// TIA Portal project "HW_2100068_montaz_menica_PSA_8HP_EL58_V18" (V18)

(* hardware
DEVICE "GSD device_8"  GSD.Device.PN
   slot 0: "vitc06a"  EX600-SPN#  EX600-SPN#
      slot 0: "EX600-SPN#"  EX600-SPN#
      slot 1: "Interface"  Interface
         slot 1: "Port 1"  Port 1
         slot 2: "Port 2"  Port 2
   slot 0: "Rack"  Rack  V1.0
   slot 1: "EX600-DX#D_1"  EX600-DX#D  EX600-DX#D
      slot 0: "EX600-DX#D"  EX600-DX#D
   slot 2: "EX600-DY#B_1"  EX600-DY#B  EX600-DY#B
      slot 0: "EX600-DY#B"  EX600-DY#B
   slot 3: "EX600-AXA_1"  EX600-AXA  EX600-AXA
      slot 0: "EX600-AXA"  EX600-AXA
   slot 4: "EX600-SPN (32 coils)_1"  EX600-SPN (32 coils)  EX600-SPN
      slot 0: "EX600-SPN"  EX600-SPN
DEVICE "GSD device_7"  GSD.Device.PN
   slot 0: "vitc04e"  EX600-SPN#  EX600-SPN#
      slot 0: "EX600-SPN#"  EX600-SPN#
      slot 1: "Interface"  Interface
         slot 1: "Port 1"  Port 1
         slot 2: "Port 2"  Port 2
   slot 0: "Rack"  Rack  V1.0
   slot 1: "EX600-DX#D_1"  EX600-DX#D  EX600-DX#D
      slot 0: "EX600-DX#D"  EX600-DX#D
   slot 2: "EX600-DY#B_1"  EX600-DY#B  EX600-DY#B
      slot 0: "EX600-DY#B"  EX600-DY#B
   slot 3: "EX600-AXA_1"  EX600-AXA  EX600-AXA
      slot 0: "EX600-AXA"  EX600-AXA
   slot 4: "EX600-SPN (32 coils)_1"  EX600-SPN (32 coils)  EX600-SPN
      slot 0: "EX600-SPN"  EX600-SPN
DEVICE "GSD device_3"  GSD.Device.PN
   slot 0: "mtstc10c"  SR-LR1  SR-LR1  1.0
      slot 0: "SR-LR1"  SR-LR1  1.0
      slot 1: "Interface"  Interface
         slot 1: "Port 1"  Port 1
   slot 0: "Rack"  Rack  V1.0
   slot 1: "Handshake and General Error Status Bits_1"  Handshake and General Error Status Bits
      slot 0: "Handshake and General Error Status Bits"  Handshake and General Error Status Bits
   slot 3: "Completion Status Bits_1"  Completion Status Bits
      slot 0: "Completion Status Bits"  Completion Status Bits
   slot 5: "Terminal Status Bits_1"  Terminal Status Bits
      slot 0: "Terminal Status Bits"  Terminal Status Bits
   slot 8: "Operation Result Status_1"  Operation Result Status
      slot 0: "Operation Result Status"  Operation Result Status
   slot 9: "Read Data 128Byte_1"  Read Data 128Byte
      slot 0: "Read Data 128Byte"  Read Data 128Byte
   slot 10: "Latch and Error Clear Control Bits_1"  Latch and Error Clear Control Bits
      slot 0: "Latch and Error Clear Control Bits"  Latch and Error Clear Control Bits
   slot 12: "Completion Clear Control Bits_1"  Completion Clear Control Bits
      slot 0: "Completion Clear Control Bits"  Completion Clear Control Bits
DEVICE "GSD device_11"  GSD.Device.PN
   slot 0: "mtstc10a"  KRC4-ProfiNet_3.2  V3.2
      slot 0: "KRC4-ProfiNet_3.2"  KRC4-ProfiNet_3.2
      slot 1: "Interface1"  Interface1
         slot 1: "Port1"  Port1
   slot 0: "Rack"  Rack  V1.0
   slot 1: "64 safe digital in- and outputs_1"  64 safe digital in- and outputs  KUKA KR C4 Device FIO64
      slot 0: "64 safe digital in- and outputs"  64 safe digital in- and outputs
   slot 2: "256 digital in- and outputs_1"  256 digital in- and outputs  KUKA KR C4 Device IO256
      slot 0: "256 digital in- and outputs"  256 digital in- and outputs
DEVICE "GSD device_18"  GSD.Device
   slot 0: "mtstc07b"  6ES7 158-0AD01-0XA0  B0
   slot 0: "Rack_0"  Rail
DEVICE "GSD device_20"  GSD.Device.PN
   slot 0: "mtstc07a"  NIC 52-RE/PNS V2.0 - V2.x  1544.100  V2.x
      slot 0: "NIC 52-RE/PNS V2.0 - V2.x"  NIC 52-RE/PNS V2.0 - V2.x
      slot 1: "PN-IO"  PN-IO
         slot 1: "Port 1"  Port 1
         slot 2: "Port 2"  Port 2
   slot 0: "Rack"  Rack  V1.0
   slot 1: "1 Unsigned32 Output_1"  1 Unsigned32 Output
      slot 0: "1 Unsigned32 Output"  1 Unsigned32 Output
   slot 2: "64 Bytes Output_1"  64 Bytes Output
      slot 0: "64 Bytes Output"  64 Bytes Output
   slot 5: "1 Unsigned32 Input_1"  1 Unsigned32 Input
      slot 0: "1 Unsigned32 Input"  1 Unsigned32 Input
   slot 6: "64 Bytes Input_1"  64 Bytes Input
      slot 0: "64 Bytes Input"  64 Bytes Input
DEVICE "GSD device_2"  GSD.Device.PN
   slot 0: "mtstc06c"  SR-LR1  SR-LR1  1.0
      slot 0: "SR-LR1"  SR-LR1  1.0
      slot 1: "Interface"  Interface
         slot 1: "Port 1"  Port 1
   slot 0: "Rack"  Rack  V1.0
   slot 1: "Handshake and General Error Status Bits_1"  Handshake and General Error Status Bits
      slot 0: "Handshake and General Error Status Bits"  Handshake and General Error Status Bits
   slot 3: "Completion Status Bits_1"  Completion Status Bits
      slot 0: "Completion Status Bits"  Completion Status Bits
   slot 5: "Terminal Status Bits_1"  Terminal Status Bits
      slot 0: "Terminal Status Bits"  Terminal Status Bits
   slot 8: "Operation Result Status_1"  Operation Result Status
      slot 0: "Operation Result Status"  Operation Result Status
   slot 9: "Read Data 128Byte_1"  Read Data 128Byte
      slot 0: "Read Data 128Byte"  Read Data 128Byte
   slot 10: "Latch and Error Clear Control Bits_1"  Latch and Error Clear Control Bits
      slot 0: "Latch and Error Clear Control Bits"  Latch and Error Clear Control Bits
   slot 12: "Completion Clear Control Bits_1"  Completion Clear Control Bits
      slot 0: "Completion Clear Control Bits"  Completion Clear Control Bits
DEVICE "GSD device_10"  GSD.Device.PN
   slot 0: "mtstc06a"  KRC4-ProfiNet_3.2  V3.2
      slot 0: "KRC4-ProfiNet_3.2"  KRC4-ProfiNet_3.2
      slot 1: "Interface1"  Interface1
         slot 1: "Port1"  Port1
   slot 0: "Rack"  Rack  V1.0
   slot 1: "64 safe digital in- and outputs_1"  64 safe digital in- and outputs  KUKA KR C4 Device FIO64
      slot 0: "64 safe digital in- and outputs"  64 safe digital in- and outputs
   slot 2: "256 digital in- and outputs_1"  256 digital in- and outputs  KUKA KR C4 Device IO256
      slot 0: "256 digital in- and outputs"  256 digital in- and outputs
DEVICE "GSD device_17"  GSD.Device
   slot 0: "mtstc05"  6ES7 158-0AD01-0XA0  B0
   slot 0: "Rack_0"  Rail
DEVICE "GSD device_16"  GSD.Device.PN
   slot 0: "mtstc04e"  KRC4-ProfiNet_3.2  V3.2
      slot 0: "KRC4-ProfiNet_3.2"  KRC4-ProfiNet_3.2
      slot 1: "Interface1"  Interface1
         slot 1: "Port1"  Port1
   slot 0: "Rack"  Rack  V1.0
   slot 1: "64 safe digital in- and outputs_1"  64 safe digital in- and outputs  KUKA KR C4 Device FIO64
      slot 0: "64 safe digital in- and outputs"  64 safe digital in- and outputs
   slot 2: "256 digital in- and outputs_1"  256 digital in- and outputs  KUKA KR C4 Device IO256
      slot 0: "256 digital in- and outputs"  256 digital in- and outputs
DEVICE "GSD device_15"  GSD.Device
   slot 0: "mtstc04b"  6ES7 158-0AD01-0XA0  B0
   slot 0: "Rack_0"  Rail
DEVICE "ET 200SP station_2"  ET 200SP-Station
   slot 0: "et200sptc10a"  IM 155-6 PN ST  6ES7 155-6AU00-0BN0  V3.3
   slot 0: "Rack_0"  Rack  6ES5 710-8MAx1
   slot 1: "111A2 DI 16x24_1"  DI 16x24VDC ST  6ES7 131-6BH00-0BA0  V1.1
      slot 1: "111A2 DI 16x24_1"  DI 16x24VDC ST
   slot 2: "111A3 DI 16x24_2"  DI 16x24VDC ST  6ES7 131-6BH00-0BA0  V1.1
      slot 1: "111A3 DI 16x24_2"  DI 16x24VDC ST
   slot 3: "112A1 DQ 16x24_1"  DQ 16x24VDC/0.5A ST  6ES7 132-6BH00-0BA0  V1.1
      slot 1: "112A1 DQ 16x24_1"  DQ 16x24VDC/0.5A ST
   slot 4: "112A2 DQ 16x24_2"  DQ 16x24VDC/0.5A ST  6ES7 132-6BH00-0BA0  V1.1
      slot 1: "112A2 DQ 16x24_2"  DQ 16x24VDC/0.5A ST
   slot 5: "112A3 DQ 16x24_3"  DQ 16x24VDC/0.5A ST  6ES7 132-6BH00-0BA0  V1.1
      slot 1: "112A3 DQ 16x24_3"  DQ 16x24VDC/0.5A ST
   slot 6: "Server module_1"  Server module  6ES7 193-6PA00-0AA0  V1.1
      slot 1: "Server module_1"  Server module
   slot 127: "BA 2xRJ45"  BA 2xRJ45  6ES7 193-6AR00-0AA0  V0.0
      slot 1: "Port_1"  X1 P1 R  6ES7 193-6AR00-0AA0  V0.0
      slot 2: "Port_2"  X1 P2 R  6ES7 193-6AR00-0AA0  V0.0
DEVICE "ET 200SP station_4"  ET 200SP-Station
   slot 0: "et200sptc06a"  IM 155-6 PN ST  6ES7 155-6AU00-0BN0  V3.3
   slot 0: "Rack_0"  Rack  6ES5 710-8MAx1
   slot 1: "111A2 DI 16x24_1"  DI 16x24VDC ST  6ES7 131-6BH00-0BA0  V1.1
      slot 1: "111A2 DI 16x24_1"  DI 16x24VDC ST
   slot 2: "111A3 DI 16x24_2"  DI 16x24VDC ST  6ES7 131-6BH00-0BA0  V1.1
      slot 1: "111A3 DI 16x24_2"  DI 16x24VDC ST
   slot 3: "112A1 DQ 16x24_1"  DQ 16x24VDC/0.5A ST  6ES7 132-6BH00-0BA0  V1.1
      slot 1: "112A1 DQ 16x24_1"  DQ 16x24VDC/0.5A ST
   slot 4: "112A2 DQ 16x24_2"  DQ 16x24VDC/0.5A ST  6ES7 132-6BH00-0BA0  V1.1
      slot 1: "112A2 DQ 16x24_2"  DQ 16x24VDC/0.5A ST
   slot 5: "112A3 DQ 16x24_3"  DQ 16x24VDC/0.5A ST  6ES7 132-6BH00-0BA0  V1.1
      slot 1: "112A3 DQ 16x24_3"  DQ 16x24VDC/0.5A ST
   slot 6: "Server module_1"  Server module  6ES7 193-6PA00-0AA0  V1.1
      slot 1: "Server module_1"  Server module
   slot 127: "BA 2xRJ45"  BA 2xRJ45  6ES7 193-6AR00-0AA0  V0.0
      slot 1: "Port_1"  X1 P1 R  6ES7 193-6AR00-0AA0  V0.0
      slot 2: "Port_2"  X1 P2 R  6ES7 193-6AR00-0AA0  V0.0
DEVICE "ET 200SP station_1"  ET 200SP-Station
   slot 0: "et200sp_111a1"  IM 155-6 PN ST  6ES7 155-6AU00-0BN0  V3.3
   slot 0: "Rack_0"  Rack  6ES5 710-8MAx1
   slot 1: "111A2 DI 16x24_1"  DI 16x24VDC ST  6ES7 131-6BH00-0BA0  V1.1
      slot 1: "111A2 DI 16x24_1"  DI 16x24VDC ST
   slot 2: "111A3 DI 16x24_2"  DI 16x24VDC ST  6ES7 131-6BH00-0BA0  V1.1
      slot 1: "111A3 DI 16x24_2"  DI 16x24VDC ST
   slot 3: "111A4 DI 16x24_3"  DI 16x24VDC ST  6ES7 131-6BH00-0BA0  V1.1
      slot 1: "111A4 DI 16x24_3"  DI 16x24VDC ST
   slot 4: "112A1 DQ 16x24_1"  DQ 16x24VDC/0.5A ST  6ES7 132-6BH00-0BA0  V1.1
      slot 1: "112A1 DQ 16x24_1"  DQ 16x24VDC/0.5A ST
   slot 5: "112A2 DQ 16x24_2"  DQ 16x24VDC/0.5A ST  6ES7 132-6BH00-0BA0  V1.1
      slot 1: "112A2 DQ 16x24_2"  DQ 16x24VDC/0.5A ST
   slot 6: "112A3 DQ 16x24_3"  DQ 16x24VDC/0.5A ST  6ES7 132-6BH00-0BA0  V1.1
      slot 1: "112A3 DQ 16x24_3"  DQ 16x24VDC/0.5A ST
   slot 7: "Server module_1"  Server module  6ES7 193-6PA00-0AA0  V1.1
      slot 1: "Server module_1"  Server module
   slot 127: "BA 2xRJ45"  BA 2xRJ45  6ES7 193-6AR00-0AA0  V0.0
      slot 1: "Port_1"  X1 P1 R  6ES7 193-6AR00-0AA0  V0.0
      slot 2: "Port_2"  X1 P2 R  6ES7 193-6AR00-0AA0  V0.0
DEVICE "GSD device_9"  GSD.Device.PN
   slot 0: "Rack"  Rack  V1.0
   slot 0: "vitc10a"  EX600-SPN#  EX600-SPN#
      slot 0: "EX600-SPN#"  EX600-SPN#
      slot 1: "Interface"  Interface
         slot 1: "Port 1"  Port 1
         slot 2: "Port 2"  Port 2
   slot 1: "EX600-DX#D_1"  EX600-DX#D  EX600-DX#D
      slot 0: "EX600-DX#D"  EX600-DX#D
   slot 2: "EX600-DY#B_1"  EX600-DY#B  EX600-DY#B
      slot 0: "EX600-DY#B"  EX600-DY#B
   slot 3: "EX600-AXA_1"  EX600-AXA  EX600-AXA
      slot 0: "EX600-AXA"  EX600-AXA
   slot 4: "EX600-SPN (32 coils)_1"  EX600-SPN (32 coils)  EX600-SPN
      slot 0: "EX600-SPN"  EX600-SPN
DEVICE "GSD device_19"  GSD.Device.PN
   slot 0: "Rack"  Rack  V1.0
   slot 0: "mtstc07b_data"  NIC 52-RE/PNS V2.0 - V2.x  1544.100  V2.x
      slot 0: "NIC 52-RE/PNS V2.0 - V2.x"  NIC 52-RE/PNS V2.0 - V2.x
      slot 1: "PN-IO"  PN-IO
         slot 1: "Port 1"  Port 1
         slot 2: "Port 2"  Port 2
   slot 1: "1 Unsigned32 Output_1"  1 Unsigned32 Output
      slot 0: "1 Unsigned32 Output"  1 Unsigned32 Output
   slot 2: "64 Bytes Output_1"  64 Bytes Output
      slot 0: "64 Bytes Output"  64 Bytes Output
   slot 5: "1 Unsigned32 Input_1"  1 Unsigned32 Input
      slot 0: "1 Unsigned32 Input"  1 Unsigned32 Input
   slot 6: "64 Bytes Input_1"  64 Bytes Input
      slot 0: "64 Bytes Input"  64 Bytes Input
DEVICE "GSD device_12"  GSD.Device.PN
   slot 0: "Rack"  Rack  V1.0
   slot 0: "mtstc07c"  NIC 52-RE/PNS V2.0 - V2.x  1544.100  V2.x
      slot 0: "NIC 52-RE/PNS V2.0 - V2.x"  NIC 52-RE/PNS V2.0 - V2.x
      slot 1: "PN-IO"  PN-IO
         slot 1: "Port 1"  Port 1
         slot 2: "Port 2"  Port 2
   slot 1: "1 Unsigned32 Output_1"  1 Unsigned32 Output
      slot 0: "1 Unsigned32 Output"  1 Unsigned32 Output
   slot 2: "64 Bytes Output_1"  64 Bytes Output
      slot 0: "64 Bytes Output"  64 Bytes Output
   slot 5: "1 Unsigned32 Input_1"  1 Unsigned32 Input
      slot 0: "1 Unsigned32 Input"  1 Unsigned32 Input
   slot 6: "64 Bytes Input_1"  64 Bytes Input
      slot 0: "64 Bytes Input"  64 Bytes Input
DEVICE "GSD device_1"  GSD.Device.PN
   slot 0: "Rack"  Rack  V1.0
   slot 1: "plc_tc04d"  PLC_tc04d  6ES7 512-1SK01-0AB0  V2.8
      slot 0: "Line_To_Cu1"  Line_To_Cu1
      slot 1: "Cu1_To_Line"  Cu1_To_Line
      slot 2: "F_Line_To_Cu1"  F_Line_To_Cu1
      slot 3: "01_SYSTEM_GENERATED_F-CD"  01_SYSTEM_GENERATED_F-CD
      slot 4: "F_CU1_To_Line"  F_CU1_To_Line
      slot 5: "02_SYSTEM_GENERATED_F-CD"  02_SYSTEM_GENERATED_F-CD
      slot 6: "Interface"  Interface
         slot 1: "Port 1"  Port 1
         slot 2: "Port 2"  Port 2
         slot 3: "Port 3"  Port 3
DEVICE "GSD device_4"  GSD.Device.PN
   slot 0: "Rack"  Rack  V1.0
   slot 1: "plc_tc08"  PLC_tc08  6ES7 512-1SK01-0AB0  V2.8
      slot 0: "Line_To_Cu1"  Line_To_Cu1
      slot 1: "Cu1_To_Line"  Cu1_To_Line
      slot 2: "F_Line_To_Cu1"  F_Line_To_Cu1
      slot 3: "01_SYSTEM_GENERATED_F-CD"  01_SYSTEM_GENERATED_F-CD
      slot 4: "F_CU1_To_Line"  F_CU1_To_Line
      slot 5: "02_SYSTEM_GENERATED_F-CD"  02_SYSTEM_GENERATED_F-CD
      slot 6: "Interface"  Interface
         slot 1: "Port 1"  Port 1
         slot 2: "Port 2"  Port 2
         slot 3: "Port 3"  Port 3
DEVICE "GSD device_21"  GSD.Device.PN
   slot 0: "Rack"  Rack  V1.0
   slot 1: "plc_tc11_cd"  PLC_tc11_cd  6ES7 512-1SK01-0AB0  V2.8
      slot 0: "Line_To_Cu1"  Line_To_Cu1
      slot 1: "Cu1_To_Line"  Cu1_To_Line
      slot 2: "F_Line_To_Cu1"  F_Line_To_Cu1
      slot 3: "01_SYSTEM_GENERATED_F-CD"  01_SYSTEM_GENERATED_F-CD
      slot 4: "F_CU1_To_Line"  F_CU1_To_Line
      slot 5: "02_SYSTEM_GENERATED_F-CD"  02_SYSTEM_GENERATED_F-CD
      slot 6: "Line_To_Cu2"  Line_To_Cu2
      slot 7: "Cu2_To_Line"  Cu2_To_Line
      slot 8: "F_Line_To_Cu2"  F_Line_To_Cu2
      slot 9: "03_SYSTEM_GENERATED_F-CD"  03_SYSTEM_GENERATED_F-CD
      slot 10: "F_CU2_To_Line"  F_CU2_To_Line
      slot 11: "04_SYSTEM_GENERATED_F-CD"  04_SYSTEM_GENERATED_F-CD
      slot 12: "Cu3_To_Line"  Cu3_To_Line
      slot 13: "Line_To_Cu3"  Line_To_Cu3
      slot 14: "Interface"  Interface
         slot 1: "Port 1"  Port 1
         slot 2: "Port 2"  Port 2
         slot 3: "Port 3"  Port 3
DEVICE "GSD device_13"  GSD.Device.PN
   slot 0: "Rack"  Rack  V1.0
   slot 1: "plcr1_110a2"  plcr1.112_X1  6ES7 516-3FN02-0AB0  V2.8
      slot 0: "Robot1_ToLine"  Robot1_ToLine
      slot 1: "LineToRobot1"  LineToRobot1
      slot 2: "Robot2_ToLine"  Robot2_ToLine
      slot 3: "LineToRobot2"  LineToRobot2
      slot 4: "Robot3_ToLine"  Robot3_ToLine
      slot 5: "LineToRobot3"  LineToRobot3
      slot 6: "Robot4_ToLine"  Robot4_ToLine
      slot 7: "LineToRobot4"  LineToRobot4
      slot 8: "LineToFLineSafety"  LineToFLineSafety
      slot 9: "FLineToLineSafety"  FLineToLineSafety
      slot 10: "TC09_ToLine"  TC09_ToLine
      slot 11: "LineToTC09"  LineToTC09
      slot 12: "Interface"  Interface
         slot 1: "Port 1"  Port 1
         slot 2: "Port 2"  Port 2
DEVICE "GSD device_14"  GSD.Device.PN
   slot 0: "Rack"  Rack  V1.0
   slot 0: "pnpn_tc11a"  PN/PN Coupler X2  6ES7 158-3AD01-0XA0  V03.00.00
      slot 0: "PN/PN Coupler X2"  PN/PN Coupler X2
      slot 1: "PN-IO-02"  PN-IO-02
         slot 1: "Port 1"  Port 1
         slot 2: "Port 2"  Port 2
   slot 1: "FDI/FDO_6Bytes/12Bytes"  IN/OUT 6 Bytes / 12 Bytes
      slot 0: "IN/OUT 6 Bytes / 12 Bytes"  IN/OUT 6 Bytes / 12 Bytes
   slot 2: "FDI/FDO_12Bytes/6Bytes"  IN/OUT 12 Bytes / 6 Bytes
      slot 0: "IN/OUT 12 Bytes / 6 Bytes"  IN/OUT 12 Bytes / 6 Bytes
   slot 3: "IN  64 Bytes"  IN  64 Bytes
      slot 0: "IN  64 Bytes"  IN  64 Bytes
   slot 4: "OUT  64 Bytes"  OUT  64 Bytes
      slot 0: "OUT  64 Bytes"  OUT  64 Bytes
   slot 5: "IN  64 Bytes_1"  IN  64 Bytes
      slot 0: "IN  64 Bytes"  IN  64 Bytes
DEVICE "pnpn_tc11b"  PnPn.Device
   slot 0: "Rack"  Rail  1.0
   slot 0: "pnpn_tc11b.X1"  PN/PN Coupler  6ES7 158-3AD10-0XA0  V4.2
   slot 1: "pnpn_tc11b.X2"  PN/PN Coupler  6ES7 158-3AD10-0XA0  V4.2
   slot 127: "BA 2xRJ45"  BA 2xRJ45  6ES7 193-6AR00-0AA0  V0.0
      slot 1: "Port_1"  X1 P1 R  6ES7 193-6AR00-0AA0  V0.0
      slot 2: "Port_2"  X1 P2 R  6ES7 193-6AR00-0AA0  V0.0
   slot 127: "BA 2xRJ45"  BA 2xRJ45  6ES7 193-6AR00-0AA0  V0.0
      slot 1: "Port_1"  X2 P1 R  6ES7 193-6AR00-0AA0  V0.0
      slot 2: "Port_2"  X2 P2 R  6ES7 193-6AR00-0AA0  V0.0
DEVICE "GSD device_43"  GSD.Device.PN
   slot 0: "Rack"  Rack  V1.0
   slot 0: "vitc11f"  EX600-SPN#  EX600-SPN#
      slot 0: "EX600-SPN#"  EX600-SPN#
      slot 1: "Interface"  Interface
         slot 1: "Port 1"  Port 1
         slot 2: "Port 2"  Port 2
   slot 1: "EX600-DX#D_1"  EX600-DX#D  EX600-DX#D
      slot 0: "EX600-DX#D"  EX600-DX#D
   slot 2: "EX600-DY#B_1"  EX600-DY#B  EX600-DY#B
      slot 0: "EX600-DY#B"  EX600-DY#B
   slot 3: "EX600-AXA_1"  EX600-AXA  EX600-AXA
      slot 0: "EX600-AXA"  EX600-AXA
   slot 4: "EX600-SPN (32 coils)_1"  EX600-SPN (32 coils)  EX600-SPN
      slot 0: "EX600-SPN"  EX600-SPN
DEVICE "GSD device_42"  GSD.Device.PN
   slot 0: "Rack"  Rack  V1.0
   slot 0: "mtstc11f"  KRC4-ProfiNet_3.2  V3.2
      slot 0: "KRC4-ProfiNet_3.2"  KRC4-ProfiNet_3.2
      slot 1: "Interface1"  Interface1
         slot 1: "Port1"  Port1
   slot 1: "64 safe digital in- and outputs_1"  64 safe digital in- and outputs  KUKA KR C4 Device FIO64
      slot 0: "64 safe digital in- and outputs"  64 safe digital in- and outputs
   slot 2: "256 digital in- and outputs_1"  256 digital in- and outputs  KUKA KR C4 Device IO256
      slot 0: "256 digital in- and outputs"  256 digital in- and outputs
DEVICE "SCALANCE W access point"  SCALANCE W-Station
   slot 0: "SCALANCE W rack"  Rail
   slot 0: "309k1_ap"  SCALANCE W 774-1 RJ45  6GK5 774-1FX00-0AA0  V6.1
DEVICE "SCALANCE XC-200"  SCALANCE X-Station
   slot 0: "SCALANCE X rack"  Rail
   slot 0: "swr1_104s1"  SCALANCE XC224  6GK5 224-0BA00-2AC2  V2.1
DEVICE "S71500/ET200MP station_1"  S7-1500 station
   slot 0: "Rail_0"  Rack  6ES7 590-1***0-0AA0
   slot 1: "plcr1_110a1"  CPU 1516F-3 PN/DP  6ES7 516-3FN01-0AB0  V2.1
      slot 3: "CPU display_1"  6ES7591-1BA00-0AA0
      slot 32768: "PROFINET interface_1"  X1
         slot 32769: "Port_1"  X1 P1
         slot 32770: "Port_2"  X1 P2
      slot 33024: "PROFINET interface_2"  X2
         slot 33025: "Port_1"  X2 P1
      slot 33280: "DP interface_1"  X3
DEVICE "GSD device_5"  GSD.Device.PN
   slot 0: "Rack"  Rack  V1.0
   slot 1: "310a1_plc.profinet interface_1"  310A1_PLC_X1  6ES7 516-3FN01-0AB0  V2.1
      slot 0: "Outputs"  Outputs
      slot 1: "Inputs"  Inputs
      slot 2: "DataToMainLine"  DataToMainLine
      slot 3: "Interface"  Interface
         slot 1: "Port 1"  Port 1
         slot 2: "Port 2"  Port 2
*)

// ===== PLC "plcr1_110a1"  CPU 1516F-3 PN/DP =====

VAR_GLOBAL   // PLC tag table "Default tag table"
   "Clock_Byte" AT %MB0 : Byte;
   "Clock_10Hz" AT %M0.0 : Bool;
   "Clock_5Hz" AT %M0.1 : Bool;
   "Clock_2.5Hz" AT %M0.2 : Bool;
   "Clock_2Hz" AT %M0.3 : Bool;
   "Clock_1.25Hz" AT %M0.4 : Bool;
   "Clock_1Hz" AT %M0.5 : Bool;
   "Clock_0.625Hz" AT %M0.6 : Bool;
   "Clock_0.5Hz" AT %M0.7 : Bool;
   "System_Byte" AT %MB1 : Byte;
   "FirstScan" AT %M1.0 : Bool;
   "DiagStatusUpdate" AT %M1.1 : Bool;
   "AlwaysTRUE" AT %M1.2 : Bool;
   "AlwaysFALSE" AT %M1.3 : Bool;
   "i_161B8_neg" AT %I381.2 : Bool;   // TC04C1_PartPresence
   "i2026.4" AT %I2026.4 : Bool;
   "iW604" AT %IW604 : Int;
   "i171B5" AT %I480.4 : Bool;
   "q_Conveyor" AT %Q1101.7 : Bool;
   "i111A3_9" AT %I483.1 : Bool;
   "i111A3_12" AT %I483.4 : Bool;
   "i2027.4" AT %I2027.4 : Bool;
   "q484.1" AT %Q484.1 : Bool;
   "q484.0" AT %Q484.0 : Bool;
   "iFrictionMoment" AT %IW2058 : Word;
   "i111A3_6" AT %I482.6 : Bool;
   "i111A3_13" AT %I483.5 : Bool;
   "q601.0" AT %Q601.0 : Bool;
   "i600.2" AT %I600.2 : Bool;
   "q384.1" AT %Q384.1 : Bool;
   "i601.1" AT %I601.1 : Bool;
   "i111A3_5" AT %I482.5 : Bool;
   "Q2900_7" AT %Q2900.7 : Bool;
   "i2026.0" AT %I2026.0 : Bool;
   "Tag_1" AT %Q134.1 : Bool;
   "ib2024" AT %IB2024 : Byte;
   "q480.0" AT %Q480.0 : Bool;
   "i2027.1" AT %I2027.1 : Bool;
   "i111A3_4" AT %I482.4 : Bool;
   "i2026.2" AT %I2026.2 : Bool;
   "i111A3_7" AT %I482.7 : Bool;
   "q384.0" AT %Q384.0 : Bool;
   "i171B1" AT %I480.0 : Bool;
   "i171B3" AT %I480.2 : Bool;
   "i111A3_3" AT %I482.3 : Bool;
   "i_161B7" AT %I380.6 : Bool;
   "q600.0" AT %Q600.0 : Bool;
   "q601.2" AT %Q601.2 : Bool;
   "Q2900_6" AT %Q2900.6 : Bool;
   "i600.0" AT %I600.0 : Bool;
   "qTC04B_OutputByte0" AT %QB500 : Byte;
   "i111A3_10" AT %I483.2 : Bool;
   "i172SB2" AT %I481.1 : Bool;
   "i601.0" AT %I601.0 : Bool;
   "Q2900_4" AT %Q2900.4 : Bool;
   "i111A3_8" AT %I483.0 : Bool;
   "ib2025" AT %IB2025 : Byte;
   "Tag_5" AT %Q1105.7 : Bool;
   "i111A3_2" AT %I482.2 : Bool;
   "Q2900_5" AT %Q2900.5 : Bool;
   "i601.3" AT %I601.3 : Bool;
   "i2027.2" AT %I2027.2 : Bool;
   "i111A3_14" AT %I483.6 : Bool;
   "i2027.0" AT %I2027.0 : Bool;
   "i111A3_0" AT %I482.0 : Bool;
   "q600.1" AT %Q600.1 : Bool;
   "i600.3" AT %I600.3 : Bool;
   "i2026.3" AT %I2026.3 : Bool;
   "i171B2" AT %I480.1 : Bool;
   "q600.2" AT %Q600.2 : Bool;
   "qRobotOutOfArea" AT %Q50.7 : Bool;
   "qTC04B_OutputByte1" AT %QB501 : Byte;
   "i171B4" AT %I480.3 : Bool;
   "i171B6" AT %I480.5 : Bool;
   "i2027.3" AT %I2027.3 : Bool;
   "i_161B7_neg" AT %I381.3 : Bool;   // TC04C2_PartPresence
   "Tag_4" AT %I451.0 : Bool;
   "iw602" AT %IW602 : Int;
   "i172SB1" AT %I481.0 : Bool;
   "i_161B8" AT %I380.7 : Bool;
   "i600.1" AT %I600.1 : Bool;
   "i2026.1" AT %I2026.1 : Bool;
   "i601.2" AT %I601.2 : Bool;
   "q482.0" AT %Q482.0 : Bool;
   "q482.1" AT %Q482.1 : Bool;
   "i111A3_15" AT %I483.7 : Bool;
   "fdi_plcr1_110a2_1byte_pnpn" AT %IB116 : Byte;   // z pnpn plcr1_110a2 :
   "iW606" AT %IW606 : Int;
   "i111A3_1" AT %I482.1 : Bool;
   "fdiEstopTC08_Profisafe" AT %I1892.0 : Bool;   // Estop TC08 -Plnenie olejom EMP
   "i111A3_11" AT %I483.3 : Bool;
   "qGreenConveyor(1)" AT %Q480.5 : Bool;
   "qRedRework(1)" AT %Q480.2 : Bool;
   "qGreenRework(1)" AT %Q480.3 : Bool;
   "qGreenConveyor" AT %Q380.5 : Bool;
   "qGreenRework" AT %Q380.3 : Bool;
   "qRedConveyor(1)" AT %Q480.4 : Bool;
   "qRedConveyor" AT %Q380.4 : Bool;
   "qRedRework" AT %Q380.2 : Bool;
END_VAR

DATA_BLOCK "Main_Safety_RTG1_DB"   // DB1, F_DB
{ S7_Optimized_Access := 'TRUE' }
NAME : FUSI
VERSION : 0.1
// stored: InstanceOfName Main_Safety_RTG1
"Main_Safety_RTG1"
BEGIN
END_DATA_BLOCK

FUNCTION_BLOCK "Main_Safety_RTG1"   // FB1, F_FBD
{ S7_Optimized_Access := 'TRUE' }
BEGIN
END_FUNCTION_BLOCK

ORGANIZATION_BLOCK "Main"   // OB1, LAD, ProgramCycle
TITLE = "Main Program Sweep (Cycle)"
{ S7_Optimized_Access := 'TRUE' }
VERSION : 0.1
   VAR_INPUT
      Initial_Call : Bool;   // Initial call of this OB
      Remanence : Bool;   // =True, if remanent data are available
   END_VAR
BEGIN
END_ORGANIZATION_BLOCK